FUNCTION_BLOCK CubicSpline//参考《数值分析》第4版李庆扬等编，p36三转角方程
VAR_INPUT
	x : ARRAY[0..4] OF LREAL;
	y : ARRAY[0..4] OF LREAL;
	dy0 : LREAL;
	dy4 : LREAL;
	xt: LREAL;
END_VAR
VAR_OUTPUT
	yt: LREAL;
	vt: LREAL;
END_VAR
VAR
	i : INT;
	h : ARRAY[0..3] OF LREAL;
	f : ARRAY[0..3] OF LREAL;
	lemda : ARRAY[0..3] OF LREAL;
	miu : ARRAY[0..3] OF LREAL;
	g : ARRAY[0..3] OF LREAL;

	//lftMat*lftVec=rghtVec，求lftVec
	lftMat : Mat3;
	lftVec : Vec3;
	rghtVec : Vec3;
	m: ARRAY[0..4] OF LREAL;
	alpha: ARRAY[0..4] OF LREAL;
	beta: ARRAY[0..4] OF LREAL;
	dAlpha: ARRAY[0..4] OF LREAL;
	dBeta: ARRAY[0..4] OF LREAL;
	tmp: LREAL;
	tmpd: LREAL;
END_VAR

FOR i:=0 TO 3 DO
	h[i] := x[i+1] - x[i];
	f[i] := (y[i+1] - y[i]) / h[i];
END_FOR

FOR i:=1 TO 3 DO
	lemda[i] := h[i] / (h[i-1] + h[i]);
	miu[i] := h[i-1] / (h[i-1] + h[i]);
	g[i] := 3 * (lemda[i] * f[i-1] + miu[i] * f[i]);
END_FOR

//才3*3，直接求逆，更大的矩阵用追赶法
lftMat := SetMat3(2,miu[1],0, lemda[2],2,miu[2], 0,lemda[3],2);
rghtVec := SetVec3(g[1]-lemda[1]*dy0, g[2], g[3]-miu[3]*dy4);
lftVec := MatMulVec(Inv3(lftMat), rghtVec);
m[0] := dy0;
FOR i:=0 TO 2 DO
	m[i+1] := lftVec.data[i];
END_FOR
m[4] := dy4;

//分段三次hermite插值
i:=0;
IF xt <= x[1] THEN//i=0
	tmp := (xt-x[i+1])/(x[i]-x[i+1]) * (xt-x[i+1])/(x[i]-x[i+1]);
	alpha[i] := tmp * (1+2*(xt-x[i])/(x[i+1]-x[i]));
	beta[i]  := tmp * (xt-x[i]);
	tmpd := (xt-x[i+1])/(x[i]-x[i+1])/(x[i]-x[i+1]);
	dAlpha[i] := tmpd * 6*(xt-x[i])/(x[i+1]-x[i]);
	dBeta[i]  := tmpd * (2*(xt-x[i])+(xt-x[i+1]));
ELSE
	alpha[i] := 0;
	beta[i]  := 0;
	dAlpha[i]:= 0;
	dBeta[i] := 0;
END_IF
FOR i:=1 TO 3 DO
	IF xt >= x[i-1] AND xt <= x[i] THEN
		tmp := (xt-x[i-1])/(x[i]-x[i-1]) * (xt-x[i-1])/(x[i]-x[i-1]);
		alpha[i] := tmp * (1+2*(xt-x[i])/(x[i-1]-x[i]));
		beta[i]  := tmp * (xt-x[i]);
		tmpd := (xt-x[i-1])/(x[i]-x[i-1])/(x[i]-x[i-1]);
		dAlpha[i] := tmpd * 6*(xt-x[i])/(x[i-1]-x[i]);
		dBeta[i]  := tmpd * (2*(xt-x[i])+(xt-x[i-1]));
	ELSIF xt >= x[i] AND xt <= x[i+1] THEN
		tmp := (xt-x[i+1])/(x[i]-x[i+1]) * (xt-x[i+1])/(x[i]-x[i+1]);
		alpha[i] := tmp * (1+2*(xt-x[i])/(x[i+1]-x[i]));
		beta[i]  := tmp * (xt-x[i]);
		tmpd := (xt-x[i+1])/(x[i]-x[i+1])/(x[i]-x[i+1]);
		dAlpha[i] := tmpd * 6*(xt-x[i])/(x[i+1]-x[i]);
		dBeta[i]  := tmpd * (2*(xt-x[i])+(xt-x[i+1]));
	ELSE
		alpha[i] := 0;
		beta[i]  := 0;
		dAlpha[i]:= 0;
		dBeta[i] := 0;
	END_IF
END_FOR
i:=4;
IF xt >= x[3] THEN
	tmp := (xt-x[i-1])/(x[i]-x[i-1]) * (xt-x[i-1])/(x[i]-x[i-1]);
	alpha[i] := tmp * (1+2*(xt-x[i])/(x[i-1]-x[i]));
	beta[i]  := tmp * (xt-x[i]);
	tmpd := (xt-x[i-1])/(x[i]-x[i-1])/(x[i]-x[i-1]);
	dAlpha[i] := tmpd * 6*(xt-x[i])/(x[i-1]-x[i]);
	dBeta[i]  := tmpd * (2*(xt-x[i])+(xt-x[i-1]));
ELSE
	alpha[i] := 0;
	beta[i]  := 0;
	dAlpha[i]:= 0;
	dBeta[i] := 0;
END_IF

yt:=0;
vt:=0;
FOR i:=0 TO 4 DO
	yt := yt + y[i]*alpha[i] + m[i]*beta[i];
	vt := vt + y[i]*dAlpha[i] + m[i]*dBeta[i];
END_FOR

END_FUNCTION_BLOCK

(* stored: Version 1.1.0.1, ProductVersion 3.1.4024.2
   POU CubicSpline: Id {c855b65d-af6d-40cf-8f6f-e563fd78b196}, SpecialFunc None *)
